{attribute 'linkalways'} 
{attribute 'no_explicit_call' := 'This FB is a CLASS and must be accessed using methods or properties'}
{attribute 'enable_dynamic_creation'}
FUNCTION_BLOCK FINAL OR_INT EXTENDS Node
VAR
	in1 : _INT(0);
	in2 : _INT(0);
	out : _INT(0);
END_VAR

METHOD PUBLIC Clone : I_Node
VAR
	pNode : POINTER TO OR_INT;
END_VAR
pNode := __NEW(OR_INT);
Clone := pNode^;
END_METHOD

METHOD FB_init : BOOL
VAR_INPUT
	bInitRetains : BOOL; // if TRUE, the retain variables are initialized (warm start / cold start)
	bInCopyCode : BOOL;  // if TRUE, the instance afterwards gets moved into the copy code (online change)
END_VAR
AddInput('in1',THIS^.in1);
AddInput('in2',THIS^.in2);
AddOutput('out', THIS^.out);
END_METHOD

METHOD PROTECTED OnExecute
VAR
END_VAR
out.Value := in1.Value OR in2.Value;
END_METHOD

END_FUNCTION_BLOCK

(* stored: Version 1.1.0.1, ProductVersion 3.1.4024.15
   POU OR_INT: Id {be7cd8b4-260d-4a60-933e-766db2ffc2d1}, SpecialFunc None
   Folder Constructor: Id {0469c378-0e51-437f-8d1e-9ec90cba3cad}
   Method Clone: Id {be0618c5-8945-4249-b747-53502f76308b}
   Method FB_init: Id {9bf925dc-71c2-4573-9220-6fe0ecaadd4d}
   Method OnExecute: Id {15c2d8ba-fd2b-4e6d-ac8b-d82be9f17bb5} *)
